// TIA Portal V18 export
// export: Created 2026-06-07T16:28:12.8579741Z, ExportSetting WithDefaults, DisplayName Totally Integrated Automation Portal, DisplayVersion V18, DisplayName TIA Portal Openness, DisplayVersion V18, DisplayName TIA Portal Version Control Interface, DisplayVersion V18, DisplayName STEP 7 Professional, DisplayVersion V18, DisplayName STEP 7 Safety, DisplayVersion V18, DisplayName WinCC Professional, DisplayVersion V18
VAR_GLOBAL   // PLC tag table "AI_Tags"
   MB_Server_NDR AT %M10.0 : Bool;   // MB_Server_NDR Modbus Tag
   MB_Server_DR AT %M10.1 : Bool;   // MB_Server_DR Modbus Tag
   MB_Server_Error AT %M10.2 : Bool;   // MB_Server_Error Modbus Tag
   MB_Server_Status AT %MW12 : Word;   // MB_Server_Status Modbus Tag
END_VAR
